Staubli VAL3: refreshStatic.pgx

program refreshStatic()
  local string l_sMenu
  local string l_sMessage
  local string l_sName
begin
  cls()
  //
  // set the view of the page..
  //
  // SET THE PAGE NUMBER
  use:nPage=150
  // USE <>PROFILE for <>PAGE
  use:nPage=use:nPage+abs(limit(saveData:mode,0,2)-2)
  // SET THE VIEW OF THE PAGE
  call language:page(l_sMenu,use:nPage)
  // define the menu
  call use:stringToArray(l_sMenu,sMenu)
  call use:setMenu(sMenu,true,3)
  call use:getMenu(sMenu,bButton)
  //
  // CREATE THE LIST
  //
  // define your list size for default
  call use:setSizeList(20,0,18,11)
  call use:setView(bLarge)
  //
  call use:listcreate("")
  //
  call use:listadd(sList)
  //
  // refresh the cursor
  use:nView=nView
  // refresh the list
  call use:listupdate(0)
  // show the tool
  call language:message(l_sMessage,124)
  call tcp:getName(l_sName,saveData:nFrameTool)
  call use:type(0,0,l_sMessage+">"+toString("",saveData:nFrameTool)+" "+saveData:tData[saveData:nFrameTool].name)
  // show the frame
  call use:type(0,1,"Frame>"+toString("",saveData:nFrameActive)+" "+saveData:fFrameItem[saveData:nFrameActive].sName)
end
